{attribute 'qualified_only'}
{attribute 'strict'}
{attribute 'to_string'}
TYPE OPC_UA_ACTION_EXECUTION_STATE :
(
	BUSY,
	DONE,
	ERROR
);
END_TYPE

(* stored: Version 1.1.0.1
   DUT OPC_UA_ACTION_EXECUTION_STATE: Id {8104fc51-85ac-0302-1679-0efdd40e2afd} *)
